// TIA Portal V18 export
// export: Created 2026-06-12T02:00:00Z, ExportSetting WithDefaults, DisplayName Totally Integrated Automation Portal, DisplayVersion V18, DisplayName TIA Portal Openness, DisplayVersion V18
TagTable "AI_B6_Tags"
  AI_B6_TICR211_Temp : Real  (PLC tag AI_B6_TICR211_Temp, HMI_Connection_1, 1 s)   // TEMP 50-80 °C
  AI_B6_TICR210_Temp : Real  (PLC tag AI_B6_TICR210_Temp, HMI_Connection_1, 1 s)   // TEMP 50-80 °C
  AI_B6_TICR201_Tank_Temp : Real  (PLC tag AI_B6_TICR201_Tank_Temp, HMI_Connection_1, 1 s)   // TEMP 50-80 °C
  AI_B6_PT201_Pressure : Real  (PLC tag AI_B6_PT201_Pressure, HMI_Connection_1, 1 s)   // PRESSURE 7-8 bar
  AI_B6_Ph201_pH : Real  (PLC tag AI_B6_Ph201_pH, HMI_Connection_1, 1 s)   // COUNT 6-8 pH
  AI_B6_ORP201_ORP : Real  (PLC tag AI_B6_ORP201_ORP, HMI_Connection_1, 1 s)   // COUNT 20-80 %
  AI_B6_DPL101_Level : Real  (PLC tag AI_B6_DPL101_Level, HMI_Connection_1, 1 s)   // LEVEL 100-500 L
  AI_B6_TICR214_Temp : Real  (PLC tag AI_B6_TICR214_Temp, HMI_Connection_1, 1 s)   // TEMP 50-80 °C
  AI_B6_TICR204_Temp : Real  (PLC tag AI_B6_TICR204_Temp, HMI_Connection_1, 1 s)   // TEMP 50-80 °C
  AI_B6_TICR205_Temp : Real  (PLC tag AI_B6_TICR205_Temp, HMI_Connection_1, 1 s)   // TEMP 50-80 °C
  AI_B6_TICR206_Temp : Real  (PLC tag AI_B6_TICR206_Temp, HMI_Connection_1, 1 s)   // TEMP 50-80 °C
  AI_B6_FHC203_Flow : Real  (PLC tag AI_B6_FHC203_Flow, HMI_Connection_1, 1 s)   // FLOW 100-200 L/h
  AI_B6_BPC201_Pressure : Real  (PLC tag AI_B6_BPC201_Pressure, HMI_Connection_1, 1 s)   // PRESSURE 7-8 bar
